TYPE ST_St030_HMI_IN_OUT ://EXTENDS ST_HMI_PL_CMD :
STRUCT
END_STRUCT
END_TYPE

(* stored: Version 1.1.0.1
   DUT ST_St030_HMI_IN_OUT: Id {a1841e73-9e57-4248-b582-3878e08d9fb4} *)
